(* IEC 61131-3 sources: Mizera_Tube/Plc (part 2) *)

(* ---- GasProp.plc ---- *)
*******************************************************************************
*   GASPROP.PLC
*   ESAutomotion
*   LASER machine - Proportional valve for cutting gas managment
*******************************************************************************
#funcdec "DynMng.plc"

VAR
#include "cnc.inc"

Appoggio:           BOOL;
KeepPropTest:       BOOL; * Prop. valve test keep
PropOutRange:       BOOL; * Gas pressure out of range
HbOutPress:         BOOL; * Hoerbiger feedback pressure out of range

PressCalcLinear:    DWORD; * Pressure calculated from linearization

AppPressCorrente:   DWORD; * Appoggio Pressione Corrente
MaxCurrPress:       DWORD; * Maximum pressure for current selected gas (mbar)
OutValvProp:        DWORD; * Prop valve setpoint pressure (mbar)
PressTol:           DWORD; * Pressure tolerance (mbar)
MinAllPressMbar:    DWORD; * Pressure min limit for alarm (mbar)
MaxAllPressMbar:    DWORD; * Pressure max limit for alarm (mbar)
TimeAlPress:        DWORD; * Delay for pressure alarm enable (ms)
ScaleBitIN:         DWORD; * Pressure input full scale in count
ScaleBitOUT:        DWORD; * Pressure output full scale in count
IA_Feedback_GAS_IN_BAR: DWORD; * Hoerbiger feedback pressure (bar)
PressMaxEvProp_APP: DWORD;

RTRIG_EnVal1:       TRIG;
RTRIG_EnVal1_G834:  TRIG;

HOERRB_CAL_REQ1     AT %SoftBtn2.10; * ANALOG HOERB CALIBRATION REQUEST BUTTON
HOERB_RESET_REQ   	AT %SoftBtn2.20; *(SoftBtn2.20) Hoerbiger reset button
TOF_RESET_HOERB:			TOF;			 * ANALOG HOERB RESET
RTRIG_RESET_HOERB:			R_TRIG;			 * ANALOG HOERB RESET REQUEST

RT_PVTST:           R_TRIG;
#defcom RT_PVTST.Q Imp. prop. valve test button
TRIG_CAL_HOERB:     TRIG; * Hoerbiger calibration request
#defcom TRIG_CAL_HOERB.Q Imp. Hoerbiger calibration request

TON_All_prop:       TON;
#defcom TON_All_prop.Q End of pressure alarm delay
TP_HOERB_CALIB:     TP;
#defcom TP_HOERB_CALIB.Q Time for Hoerbiger calibration request
TON_HOERB_CALIB2:   TON;
#defcom TON_HOERB_CALIB2.Q End delay for Hoerbiger calibration alarm
TON_FEEDBACK_GAS_IN: TON;
#defcom TON_FEEDBACK_GAS_IN.Q End of delay pressure check for Hoerbiger valve

GasCalc:           POINTS_INT_CALC;
GasCalc2:          POINTS_INT_CALC;

END_VAR

VAR_IN_OUT
#include "mem.inc"
END_VAR

#include "iol.inc"

*******************************************************************************
FUNCTION GasProp
*******************************************************************************

*******************************************************************************
*   Enable data writing
*   M300 or TstP14.14 (from TabLaser)
*******************************************************************************
CAL  RTRIG_EnVal1(CLK=EnValOut1)   ** (TstP14.14) Abilita Attuazione Valori Uscite
CAL  RTRIG_EnVal1_G834(CLK=EnValOut1_G834)   ** (TstP11.14) Abilita Attuazione Valori Uscite

LD   RTRIG_EnVal1.Q
OR   RTRIG_EnVal1_G834.Q
AND  PRGRUN_CN0                    ** M0.0 cn0.rc8.0  Programma in corso
ST   Appoggio

LD   %cn0.rc9                * Registro funzioni M canale 0
EQ   300
AND  %cn0.rc8.4              * Strobe funzioni M canale 0
OR   Appoggio
JMPCN COPYVAL

LD   %TabLsr0.L_CutPressure
ST   GasPressPgmSet                ** (LsPlc31) Gas pressure setpoint by program (mbar)

COPYVAL:

* Proportional valve type selection

LD   %config_machine4              ** LASER - Tipo gestione valv. prop. sul bus ECAT (0=DIWAL,1=HOERBIGER...)
EQ   0
AND  %config_machine2.0            ** LASER - Gestione valvola proporzionale sul bus ECAT
ST   GasPVDiwal                    ** M107.21 Cutting gas prop. valve type lanny diwal

LD   %config_machine4              ** LASER - Tipo gestione valv. prop. sul bus ECAT (0=DIWAL,1=HOERBIGER...)
EQ   1
AND  %config_machine2.0            ** LASER - Gestione valvola proporzionale sul bus ECAT
ST   GasPVHoerbiger                ** M107.22 Cutting gas prop. valve type hoerbiger

* Proportional valve test command

CAL  RT_PVTST(CLK=P_ValTestProp)   ** (LsGui18.9) Proportional valve test from setting page

LD   RT_PVTST.Q                    ** Imp. prop. valve test button
ANDN KeepPropTest                  ** Prop. valve test keep
S    KeepPropTest                  ** Prop. valve test keep
ST   Appoggio

LD   RT_PVTST.Q                    ** Imp. prop. valve test button
ANDN Appoggio
OR   PropTestRes                   ** M107.13 Proportional valve test reset from gas commands
OR   ProgRunForGas                 ** M107.10 Program running for gas managment
ORN  MACCHINA_OK                   ** M100.1  Macchina OK
OR   RESET_MACCHINA                ** M100.2  Reset macchina
R    KeepPropTest                  ** Prop. valve test keep

* Proportional valve enable conditions

LD   %config_machine29             ** Proportional valve manage only with OXYGEN
EQ   0
AND  O_O_EV_OR_ALLGAS              ** M90.15 Elettrovalvola apertura di almeno un gas
OR   O_O_EV_OPEN_O2                ** Elettrovalvola apertura Ossigeno
* La proporzionale viene disabilitata senza il ritardo alla disattivazione del program run
AND  (
LD   PRGRUN_CN0                    ** M0.0 cn0.rc8.0  Programma in corso
*ORN  ProgRunForGas                 ** M107.10 Program running for gas managment
)
OR   KeepPropTest                  ** Prop. valve test keep
OR   (
 LD   GAS_test                      ** M107.0 Test gas in progress for prop. valve
 AND  (
  LD   %config_machine29             ** Proportional valve manage only with OXYGEN
  EQ   0
      )
    )
OR  (
LD   GAS_test                      ** M107.0 Test gas in progress for prop. valve
 AND  (
   LD   %config_machine29             ** Proportional valve manage only with OXYGEN
   EQ   1
   AND  O_O_EV_OPEN_O2                ** Elettrovalvola apertura Ossigeno
   )
  )
OR   (
 LD   GAS_test
 OR   (
  LD   O_O_EV_OPEN_O2
  OR   O_O_EV_OPEN_N2
  OR   O_O_EV_OPEN_ARIA
  )
  AND  (
  LD   %config_machine29             ** Proportional valve manage only with OXYGEN
  EQ   2
 )
)
ANDN GAS_prun_close_propv
ST   GasPropEnabFromV              ** M107.23 Gas prop. valve enable from valve configuration

*******************************************************************************
* Pressure limit for selected gas
*******************************************************************************

* Pressure limit for oxygen

LD   0
ST   MaxCurrPress                  ** Maximum pressure for current selected gas (mbar)

LD   O_O_EV_OPEN_O2                ** Elettrovalvola apertura Ossigeno
JMPCN MP_OXIGEN

LD   PressMaxOssigeno              ** (rLsGui12)Pressione massima Ossigeno
ST   PressMaxEvProp_APP
ST   MaxCurrPress                  ** Maximum pressure for current selected gas (mbar)

MP_OXIGEN:

* Pressure limit for nitrogen

LD   O_O_EV_OPEN_N2                ** Elettrovalvola apertura Azoto
JMPCN MP_NITROGEN

LD   PressMaxAzoto                 ** (rLsGui13)Pressione massima Azoto
ST   MaxCurrPress                  ** Maximum pressure for current selected gas (mbar)

LD   PressMaxEvProp                ** (rLsGui11)Pressione massima valvola proporzionale
ST   PressMaxEvProp_APP

MP_NITROGEN:

* Pressure limit for cutting air

LD   O_O_EV_OPEN_ARIA              ** Elettrovalvola apertura Aria taglio
JMPCN MP_AIR

LD   PressMaxAria                  ** (rLsGui14)Pressione massima Aria
ST   MaxCurrPress                  ** Maximum pressure for current selected gas (mbar)

LD   PressMaxEvProp                ** (rLsGui11)Pressione massima valvola proporzionale
ST   PressMaxEvProp_APP

MP_AIR:

*******************************************************************************
* SETPOINT GAS PRESSURE SELECTION
*******************************************************************************
LD   0
ST   OutValvProp                   ** Prop valve setpoint pressure (mbar)

LD   GasPropEnabFromV              ** M107.23 Gas prop. valve enable from valve configuration
ANDN RETRACERUN                    ** M0.11 Ciclo di retrace in Run
JMPCN END_PRESS_UPD

* Gas pressure for Z up simulation

LD   GasEnabOnZUp                  ** M107.11 Gas enable conditions on Z up simulation
JMPCN Z_up_test

LD   %TabLsr0.L_CutPressure
ST   OutValvProp                   ** Prop valve setpoint pressure (mbar)

JMP  END_PRESS_UPD

Z_up_test:
LD   %LaserShootOn
JMPCN Z_up_test2

LD   %LsrGest0.ShootGasPress
ST   OutValvProp                   ** Prop valve setpoint pressure (mbar)

JMP  CHK_PROP_LIM

Z_up_test2:
* Gas pressure for PURGE or GAS test

LD   SPURGOrun                     ** M107.2 Gas purge in progress
JMPCN END_PURGE

LD   PressSpurgoGas                ** (rLsGui16)Pressione spurgo Gas
ST   OutValvProp                   ** Prop valve setpoint pressure (mbar)

JMP  CHK_PROP_LIM

END_PURGE:

LD   GAS_test                      ** M107.0 Test gas in progress for prop. valve
OR   KeepPropTest                  ** Prop. valve test keep
JMPCN END_PRGTST

LD   PressTestGas                  ** (rLsGui15)Pressione test Gas
ST   OutValvProp                   ** Prop valve setpoint pressure (mbar)

* Pressure limits for test/purge

CHK_PROP_LIM:

LD   OutValvProp                   ** Prop valve setpoint pressure (mbar)
GT   30000
JMPCN LIM_SUP

LD   30000
ST   OutValvProp                   ** Prop valve setpoint pressure (mbar)

JMP  LIM_INF

LIM_SUP:

LD   OutValvProp                   ** Prop valve setpoint pressure (mbar)
LT   50
JMPCN LIM_INF

LD   50
ST   OutValvProp                   ** Prop valve setpoint pressure (mbar)

LIM_INF:

* With gas valve ON, check the pressure limits for selected gas
LD   O_O_EV_OR_ALLGAS              ** M90.15 Elettrovalvola apertura di almeno un gas
JMPC CHK_PRESS_LIM

JMP  END_PRESS_UPD

END_PRGTST:

* Air pressure for APA

LD   AirEnabForAPA                 ** M107.12 Cutting air enable for APA cycle
JMPCN NoApaRun

LD   %config_machine23             ** Pressione ARIA per gestione APA
ST   OutValvProp                   ** Prop valve setpoint pressure (mbar)
JMP  END_PRESS_UPD

NoApaRun:

* Gas pressure for program execution

LD   GasPressPgmSet                ** (LsPlc31) Gas pressure setpoint by program (mbar)
ST   OutValvProp                   ** Prop valve setpoint pressure (mbar)

* Pressure limit for selected gas

CHK_PRESS_LIM:

LD   OutValvProp                   ** Prop valve setpoint pressure (mbar)
GT   MaxCurrPress                  ** Maximum pressure for current selected gas (mbar)
JMPCN END_PRESS_UPD

LD   MaxCurrPress                  ** Maximum pressure for current selected gas (mbar)
ST   OutValvProp                   ** Prop valve setpoint pressure (mbar)

END_PRESS_UPD:

LD   OutValvProp                   ** Prop valve setpoint pressure (mbar)
ST   SetOutPress                   ** (LsPlc38) Setpoint output pressure (mbar)

LD   SetOutPress                   ** (LsPlc38) Setpoint output pressure (mbar)
MUL  145                           * 14.5 PSI = 1 bar
DIV  1000
ST   SetPressPSI                   ** (LsPlc39) Setpoint output pressure (PSI*10)

********************************************************************************
* OUTPUT GAS PRESSURE COMMAND                                                  *
********************************************************************************
LD   GasPVDiwal                    ** M107.21 Cutting gas prop. valve type lanny diwal
JMPCN no_diwal_valve

LD   GAS_test                      ** M107.0 Test gas in progress for prop. valve
OR (
LD   GAS_prun                      ** M107.1 Cutting gas active from part program
ANDN GAS_prun_close_propv
)
OR   KeepPropTest                  ** Prop. valve test keep
ST   O_O_GAS_ECAT_TYPE0_ENAB       ** Enable proportional valve on bus ecat

no_diwal_valve:
LD   GasPVHoerbiger                ** M107.22 Cutting gas prop. valve type hoerbiger
OR   GasPVDiwal                    ** M107.21 Cutting gas prop. valve type lanny diwal
JMPC NoAnalogV

***************************************
*   ANALOG valve
***************************************
* Selection 12 or 16 bits output resolution

LD   BitOutValvProp                ** (rLsPlc42) Numero bit x uscita valvola prop.
EQ   0
JMPCN l11bitOut

LD   4095
ST   ScaleBitOUT                   ** Pressure output full scale in count

JMP  ComBitOut

l11bitOut:
LD   BitOutValvProp                ** (rLsPlc42) Numero bit x uscita valvola prop.
EQ   2
JMPCN l16bitOut

LD   2047
ST   ScaleBitOUT                   ** Pressure output full scale in count

JMP  ComBitOut

l16bitOut:
LD   32767
ST   ScaleBitOUT                   ** Pressure output full scale in count

ComBitOut:

NoAnalogV:
***********************************************************
* Gases Linearization
***********************************************************
LD   EnabGasOutByGraph	     			     **(rLsGui25.0) PLC option for enabling the graph (Pressure-voltage)
JMPCN NO_LINEAR

        LD   O_O_EV_OPEN_ARIA
        OR   O_O_EV_OPEN_N2
        JMPCN NO_HP_VALVE
             LD   SetOutPress                   ** (LsPlc38) Setpoint output pressure (mbar)
             ST   GasCalc2.xPercSpeed            * Speed percentual value

             LD   1
             ST   GasCalc2.xCutLineInd           * cut line index (initial value 1 to 10)

             LD   45
             ST   GasCalc2.xCodTec               * Tecnology 0=duty 1=power 2=frequency

             CAL  GasCalc2

             LD   GasCalc2.yResult               * Result
             ST   PressCalcLinear
        NO_HP_VALVE:

        LD   O_O_EV_OPEN_O2
        JMPCN ONLY_O2_VALVE
             LD   SetOutPress                   ** (LsPlc38) Setpoint output pressure (mbar)
             ST   GasCalc.xPercSpeed            * Speed percentual value

             LD   1
             ST   GasCalc.xCutLineInd           * cut line index (initial value 1 to 10)

             LD   40
             ST   GasCalc.xCodTec               * Tecnology 0=duty 1=power 2=frequency

             CAL  GasCalc

             LD   GasCalc.yResult               * Result
             ST   PressCalcLinear
        ONLY_O2_VALVE:

		 ***************************************
         *   Gas=funz(angle)
         *   #CDL
         ***************************************
         LD   PRGRUN_CN0
         ANDN PRGSTOP_CN0
         AND (
         LD   %uvHeads0.uvhCommand1
         EQ   4                              * Cutting phase
         )
         AND  %LSRPlcOp0.3
         JMPCN no_corr_gas_linear
               LD   PressCalcLinear
               ADD (
               LD   PressCalcLinear
               MULDIV(M=%TsCutDataLinear.CDL_Pressure,D=100000) * 100 %
               )
               ST   PressCalcLinear
         no_corr_gas_linear:

        *---------------------
        *   DIWAL
        *---------------------
        LD   GasPVDiwal                         ** M107.21 Cutting gas prop. valve type lanny diwal
        JMPCN NoLin1
             LD   PressCalcLinear               ** (LsPlc38) Setpoint output pressure (mbar)
             ***DIV  10000
             ST   OA_GAS_ECAT_TYPE0             ** Gas valve on bus ecat
        NoLin1:

        *---------------------
        *   HOERBIGER
        *---------------------
        LD   GasPVHoerbiger                     ** M107.22 Cutting gas prop. valve type hoerbiger
        JMPCN NoLin2
             LD   PressCalcLinear               ** (LsPlc38) Setpoint output pressure (mbar)
             ***DIV  10000
             ST   O_OA_GAS_HOERB
        NoLin2:

        *---------------------
        *   ANALOG
        *---------------------
        LD   PressCalcLinear                   ** (LsPlc38) Setpoint output pressure (mbar)
        MUL  ScaleBitOUT                   ** Pressure output full scale in count
        DIV  PressMaxEvProp_APP
        ST   OA_GAS                        ** Gas analog valve

JMP ComValv_

NO_LINEAR:

         ***************************************
         *   Gas=funz(angle)
         *   #CDL
         ***************************************
         LD   PRGRUN_CN0
         ANDN PRGSTOP_CN0
         AND (
         LD   %uvHeads0.uvhCommand1
         EQ   4                              * Cutting phase
         )
         AND  %LSRPlcOp0.3
         JMPCN no_corr_gas
              LD   PressCalcLinear
              ADD (
              LD   PressCalcLinear
              MULDIV(M=%TsCutDataLinear.CDL_Pressure,D=100000) * 100 %
              )
              ST   PressCalcLinear
         no_corr_gas:

         *---------------------
         *   DIWAL
         *---------------------
         LD   GasPVDiwal                    ** M107.21 Cutting gas prop. valve type lanny diwal
         JMPCN NoLin10
              LD   SetOutPress              ** (LsPlc38) Setpoint output pressure (mbar)
              ST   OA_GAS_ECAT_TYPE0        ** Gas valve on bus ecat
         NoLin10:
         *---------------------
         *   HOERBIGER
         *---------------------
         LD   GasPVHoerbiger                ** M107.22 Cutting gas prop. valve type hoerbiger
         JMPCN NoLin20
              LD   SetOutPress              ** (LsPlc38) Setpoint output pressure (mbar)
              ST   O_OA_GAS_HOERB
         NoLin20:

         *---------------------
         *   ANALOG
         *---------------------
         LD   SetOutPress                   ** (LsPlc38) Setpoint output pressure (mbar)
         MUL  ScaleBitOUT                   ** Pressure output full scale in count
         DIV  PressMaxEvProp_APP
         ST   OA_GAS                        ** Gas analog valve

ComValv_:

**********************************************************************
* HOERBIGER valve calibration
**********************************************************************
LD   GasPVHoerbiger                ** M107.22 Cutting gas prop. valve type hoerbiger
JMPCN NoHber

CAL  TRIG_CAL_HOERB(CLK=HOERRB_CAL_REQ) ** Hoerbiger calibration request

CAL  TP_HOERB_CALIB(IN:=TRIG_CAL_HOERB.Q, PT=7000) ** Imp. Hoerbiger calibration request

LD   TP_HOERB_CALIB.Q              ** Time for Hoerbiger calibration request
ST   O_O_CALIB_REQ_HOERB           ** Hoerbiger: calibration request

LDN  I_I_HOERBIGER_READY           ** Hoerbiger ready on bus ecat
ST   Appoggio

CAL  TON_HOERB_CALIB2(IN:=Appoggio,PT:=15000)

LD   TON_HOERB_CALIB2.Q            ** End delay for Hoerbiger calibration alarm
ST   %PLCerr7.8                   * hoerbiger calibration error

NoHber:

*------------------------------------------------------------------------------*
* CURRENT GAS PRESSURE READING
*------------------------------------------------------------------------------*

LD   GasPVDiwal                    ** M107.21 Cutting gas prop. valve type lanny diwal
JMPCN no_lanny_diwal

* Diwal valve pressure reading

LD   IA_FBACK_ECAT_TYPE0           ** Gas proportional valve feedback on bus ecat
ST   AppPressCorrente              ** Appoggio Pressione Corrente

JMP  ComValv

no_lanny_diwal:

LD   GasPVHoerbiger                ** M107.22 Cutting gas prop. valve type hoerbiger
JMPCN no_hoerbiger

* Hoerbiger valve pressure reading

LD   IA_Feedb_HOERB_GAS_OUT        ** Hoerbiger gas proportional valve feedback (OUTPUT)
ST   AppPressCorrente              ** Appoggio Pressione Corrente
JMP  ComValv

no_hoerbiger:

* Selection 12 or 16 bits input resolution

LD   BitInValvProp                 ** (rLsPlc39) Numero bit x feedback valvola prop.
EQ   0
JMPCN l16bitIn

LD   4095
ST   ScaleBitIN                    ** Pressure input full scale in count
JMP  ComBitIn

l16bitIn:

LD   BitInValvProp                 ** (rLsPlc39) Numero bit x feedback valvola prop.
EQ   1
JMPCN l16bitInFull

LD   32767
ST   ScaleBitIN                    ** Pressure input full scale in count
JMP  ComBitIn

l16bitInFull:

LD   65535
ST   ScaleBitIN                    ** Pressure input full scale in count

ComBitIn:

* Analog valve pressure reading

LD   IA_Feedback_GAS_OUT           ** Gas proportional valve feedback (OUTPUT)
MUL  PressMaxEvProp_APP
DIV  ScaleBitIN                    ** Pressure input full scale in count
ST   AppPressCorrente              ** Appoggio Pressione Corrente

LD   %config_machine29             ** Proportional valve manage only with OXYGEN
EQ   2
JMPCN AIRO2_O2_SMCS
     LD   IA_Feedback_GAS_OUT      ** (IW20)Feedback valvola proporzionale gas di taglio Output
     SUB  819
	 MUL  PressMaxEvProp_APP
     DIV  (
     LD   ScaleBitIN
     SUB  819
     )
     ST   AppPressCorrente         ** Appoggio Pressione Corrente

     * Avoid negative value visualizzation
     LD   AppPressCorrente
     LT   0
     JMPCN no_force_zero
     LD   0
     ST   AppPressCorrente
     no_force_zero:
AIRO2_O2_SMCS:

ComValv:

LD   AppPressCorrente              ** Appoggio Pressione Corrente
ST   PressCorrente                 ** (LsPlc35) Pressione Corrente (mbar)

LD   PressCorrente                 ** (LsPlc35) Pressione Corrente (mbar)
MUL  145                           * 14.5 PSI = 1 bar
DIV  1000
ST   CurPressPSI                   ** (LsPlc34) Current gas pressure (PSI*10)

****************************************************************************************************
* GAS PRESSURE OUT OF RANGE ALARM
****************************************************************************************************
LD   SetOutPress                   ** (LsPlc38) Setpoint output pressure (mbar)
MUL  FinestraAllPress              ** (rLsGui18)Finestra allarme pressione da pagina "Gas" in %
DIV  100
ST   PressTol                      ** Pressure tolerance (mbar)

LD   SetOutPress                   ** (LsPlc38) Setpoint output pressure (mbar)
ADD  PressTol                      ** Pressure tolerance (mbar)
ST   MaxAllPressMbar               ** Pressure max limit for alarm (mbar)

LD   SetOutPress                   ** (LsPlc38) Setpoint output pressure (mbar)
SUB  PressTol                      ** Pressure tolerance (mbar)
ST   MinAllPressMbar               ** Pressure min limit for alarm (mbar)

LD   MinAllPressMbar               ** Pressure min limit for alarm (mbar)
LT   0
JMPCN NoZeroMin

LD   0
ST   MinAllPressMbar               ** Pressure min limit for alarm (mbar)

NoZeroMin:

LD   PressCorrente                 ** (LsPlc35) Pressione Corrente (mbar)
GE   MinAllPressMbar               ** Pressure min limit for alarm (mbar)
AND (
LD   PressCorrente                 ** (LsPlc35) Pressione Corrente (mbar)
LE   MaxAllPressMbar               ** Pressure max limit for alarm (mbar)
)
OR   (
LD   FinestraAllPress              ** (rLsGui18)Finestra allarme pressione da pagina "Gas" in %
EQ   0
)
AND  GasPropEnabFromV              ** M107.23 Gas prop. valve enable from valve configuration
ST   PressGasOk                    ** M107.20 Gas pressure in range

LD   GasPropEnabFromV              ** M107.23 Gas prop. valve enable from valve configuration
ANDN PressGasOk                    ** M107.20 Gas pressure in range
ANDN SPURGOrun                     ** M107.2 Gas purge in progress
ST   PropOutRange                  ** Gas pressure out of range

LD   TimeMaxAllPress               ** (rLsGui19)Tempo Ritardo allarme pressione da pagina "Gas"
MUL  1000
ST   TimeAlPress                   ** Delay for pressure alarm enable (ms)

CAL  TON_All_prop(IN=PropOutRange,PT=TimeAlPress) ** Gas pressure out of range

LD   TON_All_prop.Q                ** End of pressure alarm delay
S    %PLCerr5.14                  ** PLC Err 174 Pressione valvola proporzionale fuori range

LD   RESET_ALLARMI                 ** M100.4  Cancellazione allarmi attiva
OR   Pul_Start                     ** (gPlc0.1)Start pushbutton
R    %PLCerr5.14                  ** PLC Err 174 Pressione valvola proporzionale fuori range

**********************************************************************
* Control of input gasses (AIR / O2 / N2) with Hoerbiger input valve
**********************************************************************

LD   IA_Feedback_GAS_IN_DIG        ** Hoerbiger gas proportional valve feedback (INPUT)
ST   IA_Feedback_GAS_IN_BAR        ** Hoerbiger feedback pressure (bar)

LD   O_O_EV_OR_ALLGAS              ** M90.15 Elettrovalvola apertura di almeno un gas
AND  PRGRUN_CN0                    ** M0.0 cn0.rc8.0  Programma in corso
AND  GasPVHoerbiger                ** M107.22 Cutting gas prop. valve type hoerbiger
ST   Appoggio

CAL  TON_FEEDBACK_GAS_IN(IN:=Appoggio,PT:=Delay_Press_Check) ** (rLsGui21) Delay_Press_Check

LD   MaxCurrPress                  ** Maximum pressure for current selected gas (mbar)
SUB  IA_Feedback_GAS_IN_BAR        ** Hoerbiger feedback pressure (bar)
GT   Diff_Limit_Pres               ** (rLsGui22) Input limit difference pressure
AND  TON_FEEDBACK_GAS_IN.Q         ** End of delay pressure check for Hoerbiger valve
ANDN SPURGOrun                     ** M107.2 Gas purge in progress
ST   HbOutPress                    ** Hoerbiger feedback pressure out of range

LD   HbOutPress                    ** Hoerbiger feedback pressure out of range
AND  O_O_EV_OPEN_ARIA              ** Elettrovalvola apertura Aria taglio
S    %PLCerr7.12                    ** Hoerbiger low air pressure

LD   HbOutPress                    ** Hoerbiger feedback pressure out of range
AND  O_O_EV_OPEN_N2                ** Elettrovalvola apertura Azoto
S    %PLCerr7.13                    ** Hoerbiger low nitrogen pressure

LD   HbOutPress                    ** Hoerbiger feedback pressure out of range
AND  O_O_EV_OPEN_O2                ** Elettrovalvola apertura Ossigeno
S    %PLCerr7.14                    ** Hoerbiger low oxigen pressure

LD   Pul_Reset                     ** (gPlc0.3)Reset pushbutton
OR   EMERGENZA_PLC_CN              ** M100.0  Emergenza da PLC o da CN
OR   Pul_Start                     ** (gPlc0.1)Start pushbutton
R    %PLCerr7.12                    ** Hoerbiger low air pressure
R    %PLCerr7.13                    ** Hoerbiger low nitrogen pressure
R    %PLCerr7.14                    ** Hoerbiger low oxigen pressure

LD   %PLCerr7.12                   ** Hoerbiger low air pressure
OR   %PLCerr7.13                   ** Hoerbiger low nitrogen pressure
OR   %PLCerr7.14                   ** Hoerbiger low oxigen pressure
ST   Hold_gas_refill               ** M107.24 Hoerbiger insufficient gas pressure

****************************************************************************************************
* Segnalazioni su pagina video
****************************************************************************************************

LD   GAS_test                      ** M107.0 Test gas in progress for prop. valve
OR   KeepPropTest                  ** Prop. valve test keep
AND  GasPropEnabFromV              ** M107.23 Gas prop. valve enable from valve configuration
ST   GasTestLED                    ** (LsPlc11.10) LED Comando TEST Valvola prop.

**********************************************************************
* HOERBIGER RESET
**********************************************************************

LD   HOERB_RESET_REQ			*(SoftBtn2.20) Hoerbiger reset button
ANDN %PLCmsg7.1					*Hoerbiger calibration not running
ST   Appoggio

CAL  RTRIG_RESET_HOERB(CLK=Appoggio)
CAL  TOF_RESET_HOERB(IN:=RTRIG_RESET_HOERB.Q, PT=3000)

LD   TOF_RESET_HOERB.Q
ST   O_O_HOER_RESET

END_FUNCTION

(* ---- GestAssi.plc ---- *)
*******************************************************************************
*   GESTASSI.PLC
*   ESAutomotion
*   LASER machine
*******************************************************************************
VAR
#include "Cnc.inc"

TOF_AxStop: TOF;    *Ritardo diseccitazione Assi Fermi

END_VAR

VAR_IN_OUT
#include "mem.inc"
END_VAR

#include "Iol.inc"

*******************************************************************************
*   * Gestione Segnali assi
*******************************************************************************
FUNCTION Gest_Assi

*******************************************************************************
*   Gestione segnali asse X1
*******************************************************************************
* Richiesta ordine di moto asse X1
LD   %ax27.ra3.10           * Anello di regolazione attivo
AND  %ax27.ra3.13           * Ordine di moto
ST   Ordine_Moto_X1                ** M71.0 Ordine di moto asse X1

* Moto asse X+
LD   Ordine_Moto_X1                ** M71.0 Ordine di moto asse X1
ANDN %ax27.ra3.0            * Asse fermo teorico
AND  %ax27.ra3.2            * Direzione moto asse+
ANDN AsseX1_Moto_neg               ** M71.2 Asse X1 in moto -
ST   AsseX1_Moto_pos               ** M71.1 Asse X1 in moto +

* Moto asse X-
LD   Ordine_Moto_X1                ** M71.0 Ordine di moto asse X1
ANDN %ax27.ra3.0            * Asse fermo teorico
ANDN %ax27.ra3.2            * Direzione moto asse+
ANDN AsseX1_Moto_pos               ** M71.1 Asse X1 in moto +
ST   AsseX1_Moto_neg               ** M71.2 Asse X1 in moto -

*******************************************************************************
*   Gestione segnali asse Y1
*******************************************************************************
* Richiesta ordine di moto asse Y1
LD   %ax28.ra3.10           * Anello di regolazione attivo
AND  %ax28.ra3.13           * Ordine di moto
ST   Ordine_Moto_Y1                ** M71.8 Ordine di moto asse Y1

* Moto asse Y+
LD   Ordine_Moto_Y1                ** M71.8 Ordine di moto asse Y1
ANDN %ax28.ra3.0            * Asse fermo teorico
AND  %ax28.ra3.2            * Direzione moto asse+
ANDN AsseY1_Moto_neg               ** M71.10 Asse Y1 in moto -
ST   AsseY1_Moto_pos               ** M71.9 Asse Y1 in moto +

* Moto asse Y-
LD   Ordine_Moto_Y1                ** M71.8 Ordine di moto asse Y1
ANDN %ax28.ra3.0            * Asse fermo teorico
ANDN %ax28.ra3.2            * Direzione moto asse+
ANDN AsseY1_Moto_pos               ** M71.9 Asse Y1 in moto +
ST   AsseY1_Moto_neg               ** M71.10 Asse Y1 in moto -

*******************************************************************************
*   Gestione segnali asse Z1
*******************************************************************************
* Richiesta ordine di moto asse Z1
LD   %ax29.ra3.10           * Anello di regolazione attivo
AND  %ax29.ra3.13           * Ordine di moto
ST   Ordine_Moto_Z1                ** M71.16 Ordine di moto asse Z1

* Moto asse Z+
LD   Ordine_Moto_Z1                ** M71.16 Ordine di moto asse Z1
ANDN %ax29.ra3.0            * Asse fermo teorico
AND  %ax29.ra3.2            * Direzione moto asse+
ANDN AsseZ1_Moto_neg               ** M71.18 Asse Z1 in moto -
ST   AsseZ1_Moto_pos               ** M71.17 Asse Z1 in moto +

* Moto asse Z-
LD   Ordine_Moto_Z1                ** M71.16 Ordine di moto asse Z1
ANDN %ax29.ra3.0            * Asse fermo teorico
ANDN %ax29.ra3.2            * Direzione moto asse+
ANDN AsseZ1_Moto_pos               ** M71.17 Asse Z1 in moto +
ST   AsseZ1_Moto_neg               ** M71.18 Asse Z1 in moto -

*******************************************************************************
*   Posizione sicura Asse Z per moto assi
*******************************************************************************
LD   %ax29.ra4              ** Quota asse Z
GT   %LSRCostK48            ** Valore quota sicurezza asse Z in pagina video
AND  %ax29.ra3.14           * ra3.14  Asse Z tarato
ST   Ax_Z1_posiz_OK                ** M74.7 Asse Z1 in posizione di sicurezza

LD   MACCH_IN_AUTO                 ** M100.25 SELEZIONE MACCHINA IN AUTOMATICO
ANDN PRGRUN_CN0                    ** M0.0 cn0.rc8.0  Programma in corso
OR   MACCH_IN_MANUALE              ** M100.24 SELEZIONE MACCHINA IN MANUALE
ANDN PLC_SEL_REF                   ** ui16.1 Selezione Modo REF da Plc
ANDN Ax_Z1_posiz_OK                ** M74.7 Asse Z1 in posizione di sicurezza
ST   BlcAvX1_Z1_no_OK              ** M74.2 Blocco avanz. asse X1 per Asse Z1 non posiz. OK
ST   BlcAvY1_Z1_no_OK              ** M74.5 Blocco avanz. asse Y per Asse Z non posiz. OK

LD   BlcAvX1_Z1_no_OK              ** M74.2 Blocco avanz. asse X1 per Asse Z1 non posiz. OK
AND  %ax27.ra3.13           ** X1 Ordine di moto +\-
ST   %PLCmsg4.12            ** Plc Msg 140 Blocco Asse X1:Asse Z1 non in posizione di sicurezza

LD   BlcAvY1_Z1_no_OK              ** M74.5 Blocco avanz. asse Y per Asse Z non posiz. OK
AND  %ax28.ra3.13           * Y1 Ordine di moto +\-
ST   %PLCmsg4.16            ** Plc Msg 144 Blocco Asse Y1:Asse Z1 non in posizione di sicurezza

*******************************************************************************
*   Blocco Avanzamento X1/Y1: Sensore capacitivo in contatto con la lamiera
*******************************************************************************
LD   %PLCerr5.4             **PLC Err 164 Tip touch (A11=1, A14=0, A15=0 in normal operation)
OR   %PLCerr5.5             **PLC Err 165 Body touch (A11=1, A14=1, A15=0 in normal operation)
ANDN GEN_REF_RUN                   ** M100.16 Ciclo di Reference GENERALE in corso
ST   BlcAvX1_Sens_Capac            ** M74.3 Blocco avanz. asse X1 Sens. Capacitivo in contatto con la lamiera
ST   BlcAvY1_Sens_Capac            ** M74.6 Blocco avanz. asse Y Sens. Capacitivo in contatto con la lamiera

*******************************************************************************
*   Blocco avanzamento X1/Y1
*******************************************************************************
LD   BL_AV_ASSI_X_OVR              ** M74.8 Blocco avanzamento assi dopo Override=0 o NC_STOP
ANDN PRGSTOP_CN0                   ** (cn0.rc8.1)  Programma interrotto CN0
OR   BlcAvX1_Z1_no_OK              ** M74.2 Blocco avanz. asse X1 per Asse Z1 non posiz. OK
OR   BlcAvX1_Sens_Capac            ** M74.3 Blocco avanz. asse X1 Sens. Capacitivo in contatto con la lamiera
OR   BlcAvY1_Sens_Capac            ** M74.6 Blocco avanz. asse Y Sens. Capacitivo in contatto con la lamiera
ST   BlcAvX1_user                  ** M74.0 Blocco avanzamento asse X1 da user.plc
ST   BlcAvY1_user                  ** M74.4 Blocco avanzamento asse Y da user.plc

****************************************************************************************************
*   Segnale Assi Fermi
****************************************************************************************************
CAL  TOF_AxStop(IN=AxStopSincGRP,PT=50) ** Ritardo diseccitazione Assi Fermi

LD   TOF_AxStop.Q
ST   AxStop_ForUser                ** (gPlc13.14) Info Assi fermi a User

END_FUNCTION

(* ---- IOConfig.plc ---- *)
*******************************************************************************
*   IOCONFIG.PLC
*   ESAutomotion
*   LASER machine
*******************************************************************************
#funcdec "res_ipg.plc"
#funcdec "LsrGest.plc"
#funcdec "CAP_Prec.plc"
#funcdec "FocProco.plc"

VAR
#include "Cnc.inc"
#include "Iof.inc"       * I/O Applicativo
END_VAR

VAR_IN_OUT
#include "mem.inc"
END_VAR

#include "Iol.inc"
#include "res_ipg.inc"
#include "LsrGest.inc"
#include "Cap_Prec.inc"
#include "foc_prec.inc"
#include "Aspiraz.inc"
#include "nLight.inc"

*#include "zVar.inc"

VAR
TM_offLSR:                       TOF;
TM_OnLSR:                        TON;
TM_StartButton:                   TP;
AppStartLSR:                    BOOL;
GuardDoorAutoUp:                BOOL;
GuardDoorAutoDwn:               BOOL;
RTRIG_A1_LASER_REQ:           R_TRIG;
TOF_A1_LASER_REQ:                TOF;

TP_Fence:                         TP;
FTRIG_Fence:                  F_TRIG;
R_TRIG_Door_Up_Gui_1:         R_TRIG;
R_TRIG_Door_Down_Gui_1:       R_TRIG;
R_TRIG_Door_Up_Gui_2:         R_TRIG;
R_TRIG_Door_Down_Gui_2:       R_TRIG;
END_VAR

*******************************************************************************
*   I/O CONFIGURATION (INPUT)
*******************************************************************************
FUNCTION INP_CONFIG

***************************************
*   GENERIC
***************************************
LDN  I_EMERGENZA
S    I_I_EMERGENZA               * Machine OK (no EMERG.)

LD   Pul_Reset
R    I_I_EMERGENZA

LD   I_CHILLER_ERR				* Chiller error
ANDN %LSRPlcOp0.8
ST   I_I_CHILLER_ERR
ST   %PLCerr6.0

LD   I_ASPIRATORE_OK
ST   I_I_ASPIRATORE_OK

***
*** *Comandi operatore
*** *----------------------------
LD  I_PUL_START
ST  I_I_PUL_START               * Start
LD  I_PUL_STOP
ST  I_I_PUL_STOP                * Stop
LD  I_PUL_RESET
ST  I_I_PUL_RESET               * Reset
***
*** *Hold macchina
*** *----------------------------
***  LD  M_HoldAlarmMac              *Hold macchina per allarme
***  ST  CMD_HOLD_MAC                * M206.0 Hold (CH0, CH3)
***
*** *Hold assi
*** *----------------------------
***  LD  M_HoldAx_X
***  ST  CMD_HOLDMOVING_CH3.0
***  LD  M_HoldAx_Y
***  ST  CMD_HOLDMOVING_CH3.1
***  LD  M_HoldAx_Z
***  ST  CMD_HOLDMOVING_CH3.2
*** LD  M_HoldAx_U
*** ST  CMD_HOLDMOVING_CH3.3
***  LD  M_HoldAx_B
***  ST  CMD_HOLDMOVING_CH3.7
***  LD  M_HoldAx_Cm
***  ST  CMD_HOLDMOVING_CH3.8
***
***  LD  M_HoldAx_Cs
***  ST  CMD_HOLDMOVING_CH5.8

 *Drives ok
 *----------------------------

*************************************************
*   GAS
*************************************************
 *Ingresso analogica
 *----------------------------
  LD  %ecat_ring0.EcatNode20.EcMDPIn1
  ST  IA_FBACK_ECAT_TYPE0

 *Ingresso digitale
 *----------------------------
  LD  I_PRESSIONE_ARIA_IMPIANTO
  ST  I_I_PRESSIONE_ARIA_IMPIANTO * Pressione aria Impianto OK

  LD  I_PRESSIONE_N2
  ST  I_I_PRESSIONE_N2            * Pressione Azoto OK

  LD  I_PRESSIONE_O2
  ST  I_I_PRESSIONE_O2            * Pressione Ossigeno OK

  LD  I_PRESSIONE_ARIA
  OR(
   LD %rLsGui14
   LE 0
  )
  ST  I_I_PRESSIONE_ARIA          * Pressione Aria di taglio OK

  LD  I_PRESSIONE_ARIA_BANCO      * PLCFLAGS.1  Flag sempre stato on
  ST  I_I_PRESSIONE_ARIA_BANCO    * Pressione aria Banco OK

* HOERBIGER VALVE

LD   I_IA_Feedb_HOERB_GAS_OUT
ST   IA_Feedb_HOERB_GAS_OUT       * Hoerbiger gas proportional valve feedback (OUTPUT)

LD   I_HOERBIGER_READY          * Hoerbiger ready on bus ecat
ST   I_I_HOERBIGER_READY          * Hoerbiger ready on bus ecat

*************************************************
*   RESONATOR (IPG)
*************************************************
PATH %Resonator[0]
PATH %LsrGest[0]

* Gestione laser IPG YSL
***************************************
LD   %config_machine28
EQ   0
JMPCN NoLSR_IPG_YLS

 *Ingressi digitali
 *----------------------------
  LD   I_LSR_READY
  ST   I_B1_LASER_READY           ** IPG Laser internal main power supply ON (Aux Power ON)

  LD   I_LSR_WARNING
  ST   I_B13_AVVERTENZA           ** IPG WARNING OUT

  LD   I_LSR_ERROR
  ST   I_B4_LASER_ERROR           ** IPG YLS YLR Laser in Alarm status

  LD   I_LSR_GUIDE_ON
  ST   I_B5_LASER_GUIDE           ** IPG Laser guida ON

  LD   I_LSR_EMISSION_ON
  ST   I_B2_EMISSION_ON           ** IPG Emission ON

  LD   ALWAYS_ONE
  ST   I_B7_LASER_ASSIGNED        ** IPG Laser ASSIGNED

  LD   ALWAYS_ONE
  ST   I_B8_POWER_SUPPLY          ** IPG power supply status

  LD   ALWAYS_ONE
  ST   I_B6_ANALOG_CONTROL        ** IPG Controllo analogico ON

***************************************
NoLSR_IPG_YLS:

*Gestione laser IPG YSR - RACK
***************************************
LD   %config_machine28
EQ   1
JMPCN NoLSR_IPG_YLR

 *Ingressi digitali
 *----------------------------
  LD   %PLCFLAGS.1
  ST   I_B1_LASER_READY              ** IPG Laser internal main power supply ON (Aux Power ON)

  LDN  I_LSR_READY
  AND  I_LSR_LASER_ON
  ST   I_B4_LASER_ERROR              ** IPG YLS YLR Laser in Alarm status

  LD   I_LSR_EMISSION_ON
  ST   I_B2_EMISSION_ON              ** IPG Emission ON

  LD   %PLCFLAGS.1
  ST   I_B7_LASER_ASSIGNED           ** IPG Laser ASSIGNED

  LD   ALWAYS_ONE
  ST   I_B8_POWER_SUPPLY             ** IPG power supply status

 *Ingressi simulati
 *----------------------------
  LD   %PLCFLAGS.0
  ST   I_B13_AVVERTENZA              ** IPG WARNING OUT

  LD   O_A6_ANALOG_CONTROL
  AND  I_B8_POWER_SUPPLY             ** IPG power supply status
  ST   I_B6_ANALOG_CONTROL           ** IPG Controllo analogico ON

  LD   O_A5_GUIDE_LASER
  AND  I_B8_POWER_SUPPLY             ** IPG power supply status
  ST   I_B5_LASER_GUIDE              ** IPG Laser guida ON

 *SEGNALI NON GESTITI
 *----------------------------
  *I_B3_INT_CONTROL              ** IPG Controllo interno abilitato

***************************************
NoLSR_IPG_YLR:

LD   %config_machine28
EQ   2
JMPCN LSR_RAYCUS
      LD   I_LSR_READY
      ST   I_B1_LASER_READY              ** IPG Laser internal main power supply ON (Aux Power ON)

      LD   %PLCFLAGS.1
      ST   I_B7_LASER_ASSIGNED           ** IPG Laser ASSIGNED

	  LD   I_LSR_EMISSION_ON
      ST   I_B2_EMISSION_ON              ** IPG Emission ON

      LD   I_LSR_ASSIGNED
      ST   I_B8_POWER_SUPPLY             ** IPG power supply status

      LD   I_LSR_ERROR
      ST   I_B4_LASER_ERROR           ** IPG YLS YLR Laser in Alarm status
LSR_RAYCUS:

**************************************************
* nLight Resonator Management

PATH %Resonator[1]
PATH %LsrGest[0]

LD   %config_machine28
EQ   5
JMPCN no_nlight_resonator

LD   I_FW_READY_nLight
ST   I_I_FW_READY_nLight                     * NLIGHT: nLight ready to recieve input

LD   I_EMISS_nLight
ST   I_I_EMISS_nLight                        * NLIGHT: emiss nlight enable

LD   I_ERR_nLight
ST   I_I_ERR_nLight                          * NLIGHT: nlight error

LD   I_RDY_nLight
ST   I_I_RDY_nLight                          * NLIGHT: laser nlight ready

LD   I_ExtCtr_Ready_nLight
ST   I_I_ExtCtr_Ready_nLight                 * NLIGHT: nLight external control ready

no_nlight_resonator:

*************************************************
*   CAPACITIVE
*************************************************
PATH %Capacitive[0]

* Ingressi analogica
*----------------------------
* mainfast.plc
* LD   I_PREC_CAPACITIVO
* ST   IA_A18_19_DIST_LINEAR      * Capacitive sensor

* Ingressi digitali
*----------------------------

LD   %config_machine26
EQ   4
JMPC PREC_IO_TYPE

     LD   I_PREC_FAR
     ST   I_FAR_A10                  ** Far away

     LD   I_PREC_COLLISION
     ST   I_TIP_BODY_TOUCH_A11       ** Tip\Body Touch or Nozzle_Lost (TIP TOUCH:A11=1,A14=0,A15=0)

     LD   I_PREC_BROKEN
     ST   I_CABLE_CUT_A12            ** Cable cut

     LD   I_PREC_READY
     ST   I_READY_A13                ** Ready

     LD   I_PREC_BODY_TOUCH
     ST   I_BODY_TOUCH_A14           ** Body touch (A11=1,A14=1,A15=0)

     LD   I_PREC_REACH
     ST   I_NOZZLE_LOST_A15          ** Nozzle Lost/Pos reached (NOZZLE LOST:A11=1,A14=0,A15=1)

PREC_IO_TYPE:

LD   %config_machine26
EQ   4
JMPCN PREC_LIKE_ECAT

     LD   I_ECAT_FAR
     ST   I_FAR_A10                  ** Far away

     LD   I_ECAT_COLLISION
     ST   I_TIP_BODY_TOUCH_A11       ** Tip\Body Touch or Nozzle_Lost (TIP TOUCH:A11=1,A14=0,A15=0)

     LD   I_ECAT_BROKEN
     ST   I_CABLE_CUT_A12            ** Cable cut

     LD   I_ECAT_READY
     ST   I_READY_A13                ** Ready

     LD   I_ECAT_BODY_TOUCH
     ST   I_BODY_TOUCH_A14           ** Body touch (A11=1,A14=1,A15=0)

     LD   I_ECAT_REACH
     ST   I_NOZZLE_LOST_A15          ** Nozzle Lost/Pos reached (NOZZLE LOST:A11=1,A14=0,A15=1)

PREC_LIKE_ECAT:

*************************************************
*   LENS
*************************************************
PATH %Head_Laser[0]

*Gestione focale PRECITEC
***************************************
LD   %config_machine25
EQ   0
JMPCN NoLENS_PREC

  LDN  I_PREC_ERROR
  ST   I_I_PREC_ERROR                ** precitec in error

  LD   I_PREC_INPOS
  ST   I_I_PREC_POSITION_REACHED     ** Position Reached
***************************************
NoLENS_PREC:

END_FUNCTION

*******************************************************************************
*   I/O CONFIGURATION (OUTPUT)
*******************************************************************************
FUNCTION OUT_CONFIG

*************************************************
*   GENERIC
*************************************************
 *Uscite digitali
 *----------------------------
  LD  O_O_CNC_OK                  * CNC OK
  ST  O_CN_READY

 * LD  ALARM_ACT		         ** M100.3  Allarme attivo
 * ST  AlarmExt                    * Allarmi Esterno

* Hoerbiger Valve

*LD   O_O_ENAB_VALVE_HOERB
*ST   O_ENAB_VALVE_HOERB

LD   O_O_PILOT_HOERB
ST   O_PILOT_HOERB

LD   O_O_CALIB_REQ_HOERB
ST   O_CALIB_REQ_HOERB

LD   O_O_EV_OPEN_N2_HOERB
ST   O_EV_OPEN_N2_HOERB

LD   O_O_EV_OPEN_O2_HOERB
ST   O_EV_OPEN_O2_HOERB

LD   O_O_EV_OPEN_ARIA_HOERB
ST   O_EV_OPEN_ARIA_HOERB

*LD   O_O_GAS_ECAT_TYPE0_ENAB
*ST   O_GAS_ECAT_TYPE0_ENAB

LD   O_OA_GAS_HOERB
ST   OA_GAS_HOERB

*************************************************
*   GAS
*************************************************
 *Uscite analogica
 *----------------------------
 * LD  OA_GAS_ECAT_TYPE0           * Uscita Valvola Proporzionale Gas di taglio
 * ST  %ecat_ring0.EcatNode16.EcMDPOut1

 * LD  O_O_GAS_ECAT_TYPE0_ENAB     * Abilita Valvola Proporzionale
 * ST  %ecat_ring0.EcatNode16.EcMDPOut0.0

 *Uscite digitali
 *----------------------------
  LD  O_O_EV_ARIA_UGELLO         * Elettrovalvola aria ugello
  ST  O_EV_ARIA_UGELLO

  LD  O_O_EV_OPEN_ARIA           * Elettrovalvola apertura Aria taglio
  ST  O_EVGAS_ARIA

  LD  O_O_EV_OPEN_N2             * Elettrovalvola apertura Azoto
  ST  O_EVGAS_OAZOTO

  LD  O_O_EV_OPEN_O2             * Elettrovalvola apertura Ossigeno
  ST  O_EVGAS_OSSIGENO

  LD  O_O_EV_AUX_GAS             * Elettrovalvola ausiliaria (a valle della proporzionale)
  ST  O_EV_AUX_GAS

  LD  O_EVGAS_ARIA
  OR  O_EVGAS_OAZOTO
  OR  O_EVGAS_OSSIGENO
  ST  O_EVGAS_PRES                * Output pressurizzazione gas

 *SEGNALI NON GESTITI
 *----------------------------
  *O_O_EV_ASSISTENZA_TAGLIO      * Elettrovalvola assistenza taglio

*************************************************
*   RESONATOR
*************************************************
PATH %Resonator[0]
PATH %LsrGest[0]

*Gestione laser IPG YSL
***************************************
LD   %config_machine28
EQ   0
JMPCN NoLSR_IPG_YLS

 *Gestione yEmission direttamente su scheda PWM
 *----------------------------
 LD  OUT_isFlyCutModeON            * IN "FLYCUT" or M851 cannot write on this register
 JMPC YLS_FlyCut
  LD   O_A1_LASER_REQ             ** IPG Richiesta Laser
  ST   %QW911.8

  CAL  RTRIG_A1_LASER_REQ(CLK:=O_A1_LASER_REQ)
  CAL  TOF_A1_LASER_REQ(IN=RTRIG_A1_LASER_REQ.Q,PT=1000)

  LD   TOF_A1_LASER_REQ.Q
  ST   O_LSR_REQUEST
 YLS_FlyCut:

 *Uscite digitali
 *----------------------------
  LD   O_C1_LASER_SWITCH          ** IPG Laser Switch ON
  ST   O_LSR_LASER_ON

  LD   O_A4_LASER_RESET           ** IPG Resetta errori
  ST   O_LSR_RESET

  LD   O_A5_GUIDE_LASER           ** IPG Laser spot guide ON
  ST   O_LSR_GUIDE_ON

  LD   O_A6_ANALOG_CONTROL        ** IPG Controllo analogico ON
  ST   O_LSR_ANALOG_CONTROL

***************************************
NoLSR_IPG_YLS:

*Gestione laser IPG YSR - RACK
***************************************
LD   %config_machine28
EQ   1
JMPCN NoLSR_IPG_YLR

 *Gestione Remote start (solo IPG Rack)
 *----------------------------
  *Gestione fronte di salita
  *I_LSR_WORNING è collegato Laser PS Active Pin 5-7 conn.EMG)
*  CAL TM_OnLSR(IN=AuxOn,PT=500)
*  LD   TM_OnLSR.Q
*  AND  O_A1_LASER_REQ                ** IPG Richiesta Laser
*  ST   AppStartLSR
*  CAL  TM_StartButton(IN=AppStartLSR,PT=1500)

*  LD   TM_StartButton.Q
*  ST   O_LSR_REMOTE_START

 *Uscite digitali
 *----------------------------
  LD   O_A4_LASER_RESET           * IPG Resetta errori
  ST   O_LSR_RESET

  LD   O_A5_GUIDE_LASER           * IPG Laser spot guide ON
  ST   O_LSR_GUIDE_ON

***************************************
NoLSR_IPG_YLR:

LD   %config_machine28
EQ   2
JMPCN LSR_RAYCUS_OUT
      LD   O_A5_GUIDE_LASER           * IPG Laser spot guide ON
      ST   O_LSR_GUIDE_ON

      LD   O_A1_LASER_REQ
      ST   O_LSR_LASER_ON

	  LD   O_C1_LASER_SWITCH
	  ST   O_LSR_REMOTE_START

	  LD   O_A4_LASER_RESET           ** IPG Resetta errori
      ST   O_LSR_RESET

	  * Some models of Raycus needs to add delay with fc-out (Laser Enable)
	  * In such a case, it requires to use pure PWM control and FcOut always 1
	  LD   PAR_combinedMode
	  JMPCN RAY_PUREPWM
	       LD   O_A1_LASER_REQ             ** IPG Richiesta Laser
           ST   %QW911.8
	  RAY_PUREPWM:
LSR_RAYCUS_OUT:

**************************************************
* nLight Resonator Management

PATH %Resonator[1]
PATH %LsrGest[0]

LD   %config_machine28
EQ   5
JMPCN no_nlight_resonator1

LD   O_O_EXTEN_IN_nLight                   * NLIGHT: nlight exten in
ST   %M5.0

LD   O_O_GUIDE_nLight                      * NLIGHT: Guide laser nlight
ST   O_LSR_GUIDE_ON

*LD   O_O_SYSTEM_ON_nLight                  * NLIGHT: nlight system on
*ST   %QW3.3

LD   O_O_RESET_nLight                      * NLIGHT: reset error nlight
ST   O_LSR_RESET

LD   O_O_ExtCtr_ENABLE_nLight              * NLIGHT: Enable external control of nlight
ST   %M5.0

no_nlight_resonator1:

*************************************************
*   CAPACITIVE
*************************************************
PATH %Capacitive[0]
 *Uscite digitali
 *----------------------------

LD   %config_machine26
EQ   4
JMPC PREC_IO_TYPE_OUT

     LD  O_CALIBRA_REQ_A3            * Calibration request
     ST  O_PREC_CALIBRAZIONE

     LD  O_STROBE_A7                 * Strobe
     ST  O_PREC_STROBE

     LD  O_SELCHAR_BIT0_A4           * Selecting the calibrated characteristic curve (1-8)
     ST  O_PREC_SELCHAR_0

     LD  O_SELCHAR_BIT1_A5           * Selecting the calibrated characteristic curve (1-8)
     ST  O_PREC_SELCHAR_1

     LD  O_SELCHAR_BIT2_A6           * Selecting the calibrated characteristic curve (1-8)
     ST  O_PREC_SELCHAR_2

PREC_IO_TYPE_OUT:

LD   %config_machine26
EQ   4
JMPCN PREC_LIKE_ECAT_OUT

     LD  O_CALIBRA_REQ_A3            * Calibration request
     ST  O_ECAT_CALIBRAZIONE

     LD  O_STROBE_A7                 * Strobe
     ST  O_ECAT_STROBE

     LD  O_SELCHAR_BIT0_A4           * Selecting the calibrated characteristic curve (1-8)
     ST  O_ECAT_SELCHAR_0

     LD  O_SELCHAR_BIT1_A5           * Selecting the calibrated characteristic curve (1-8)
     ST  O_ECAT_SELCHAR_1

     LD  O_SELCHAR_BIT2_A6           * Selecting the calibrated characteristic curve (1-8)
     ST  O_ECAT_SELCHAR_2

PREC_LIKE_ECAT_OUT:

*************************************************
*   LENS
*************************************************
PATH %Head_Laser[0]

*Gestione focale PRECITEC
***************************************
LD   %config_machine25
EQ   0
JMPCN NoLENS_PREC

  LD   O_O_PREC_AUTOMATIC         * Automatic request fo precitec head
  ST   O_PREC_POSITION

  LD   O_O_PREC_REFERENCE         * Reference signal for precitec head
  ST   O_PREC_REF

  LD   OA_FOCALE                  * Focal analog out
  ST   O_PREC_FOCALE

***************************************
NoLENS_PREC:

*************************************************
*   Clamp
*************************************************

LD   O_O_CLAMP_C_CLOSE           *AT %M62.9;
ST   O_CLAMP_C_CLOSE

LD   O_O_CLAMP_C_OPEN           *AT %M62.10;
ST   O_CLAMP_C_OPEN

LD   O_O_CLAMP_C1_CLOSE           *AT %M62.11;
ST   O_CLAMP_C1_CLOSE

LD   O_O_CLAMP_C1_OPEN           *AT %M62.12;
ST   O_CLAMP_C1_OPEN

*************************************************
*   MACHINE LIGHT
*************************************************
LD   O_O_LUCE_CABINA          * AT %M60.0;
ST   O_LUCE_CABINA

LD   O_O_LAMPADA_ROSSA
ST   O_LAMPADA_ROSSA

LD   O_O_LAMPADA_ROSSA
AND  %PLCFLAGS.10
ANDN %LSRPlcOp1.27
ST   O_BUZZER_ALARM

LD   O_O_LAMPADA_ARANCIONE
ST   O_LAMPADA_ARANCIONE

LD   O_O_LAMPADA_VERDE
ST   O_LAMPADA_VERDE

LD   O_O_BUZZER_START_CIC
ST   O_BUZZER_START_CIC

*************************************************
*   Lubrication
*************************************************
LD   I_LUB_LOW_LEVEL
ST   I_I_LUB_LOW_LEVEL        *AT %M55.5;

LD   I_LUB_LOW_PRESSURE
ST   I_I_LUB_LOW_PRESSURE     *AT %M55.9;

LD   I_OVER_PRES_LUB
ST   I_I_OVER_PRES_LUB        *AT %M55.10

LD   O_O_LUB                  *AT %M60.7;
ST   O_LUB

*************************************************
*   ASPIRATORE
*************************************************

LD   O_START_ASPIRATORE        *AT %DigOutAspirator1.0  Command START for Aspiration system
ST   START_ASPIRATORE
ST   START_ASPIRATORE_FUMI

*************************************************
*   Limit Switch
*************************************************

LD   I_FC_Y1_POS
ST   I_I_FC_Y1_POS        *AT %M53.2;

LD   I_FC_Y1_NEG
ST   I_I_FC_Y1_NEG        *AT %M53.3;

LD   I_FC_X1_POS
ST   I_I_FC_X1_POS        *AT %M53.0;

LD   I_FC_X1_NEG
ST   I_I_FC_X1_NEG        *AT %M53.1;

LD   I_FC_Z1_POS
ST   I_I_FC_Z1_POS        *AT %M53.4;

LD   I_FC_Z1_NEG
ST   I_I_FC_Z1_NEG        *AT %M53.5;

LD   I_FC_UV_POS
ST   I_I_FC_UV_POS        *AT %M53.6;

LD   I_FC_UV_NEG
ST   I_I_FC_UV_NEG        *AT %M53.7;

LD   I_FC_W1_POS
ST   I_I_FC_W1_POS        *AT %M53.8;

LD   I_FC_W1_NEG
ST   I_I_FC_W1_NEG        *AT %M53.9;

LD   I_FC_V_POS
ST   I_I_FC_V_POS         *AT %M53.18;

LD   I_FC_V_NEG
ST   I_I_FC_V_NEG         *AT %M53.19;

LD   I_FC_Z1_SUP_NEG
ST   I_I_FC_Z1_SUP_NEG

LD   I_FC_Z2_SUP_NEG
ST   I_I_FC_Z2_SUP_NEG

LD   I_FC_Z3_SUP_NEG
ST   I_I_FC_Z3_SUP_NEG

LD   I_FC_Z4_SUP_NEG
ST   I_I_FC_Z4_SUP_NEG

LD   I_FC_Z1_SUP_POS
ST   I_I_FC_Z1_SUP_POS

LD   I_FC_Z2_SUP_POS
ST   I_I_FC_Z2_SUP_POS

LD   I_FC_Z3_SUP_POS
ST   I_I_FC_Z3_SUP_POS

LD   I_FC_Z4_SUP_POS
ST   I_I_FC_Z4_SUP_POS

LD   I_FC_L1_NEG
ST   I_I_FC_L1_NEG

LD   I_FC_L2_NEG
ST   I_I_FC_L2_NEG

LD   I_FC_L3_NEG
ST   I_I_FC_L3_NEG

LD   I_FC_L4_NEG
ST   I_I_FC_L4_NEG

LD   I_FC_L5_NEG
ST   I_I_FC_L5_NEG

LD   I_FC_L1_POS
ST   I_I_FC_L1_POS

LD   I_FC_L2_POS
ST   I_I_FC_L2_POS

LD   I_FC_L3_POS
ST   I_I_FC_L3_POS

LD   I_FC_L4_POS
ST   I_I_FC_L4_POS

LD   I_FC_L5_POS
ST   I_I_FC_L5_POS

LD   I_FC_O4_POS
ST   I_I_FC_O4_POS
LD   I_FC_O3_POS
ST   I_I_FC_O3_POS
LD   I_FC_O2_POS
ST   I_I_FC_O2_POS
LD   I_FC_O1_POS
ST   I_I_FC_O1_POS

LD   I_FC_O4_NEG
ST   I_I_FC_O4_NEG
LD   I_FC_O3_NEG
ST   I_I_FC_O3_NEG
LD   I_FC_O2_NEG
ST   I_I_FC_O2_NEG
LD   I_FC_O1_NEG
ST   I_I_FC_O1_NEG

LD   I_FC_W_NEG
ST   I_I_FC_W_NEG
LD   I_FC_W_POS
ST   I_I_FC_W_POS

LD   I_FC_B1_POS
ST   I_I_FC_B1_POS
LD   I_FC_B1_NEG
ST   I_I_FC_B1_NEG

LDN  I_AntiColide_1
ORN  I_AntiColide_2
ST   I_I_AntiColide
S    %PLCerr21.24

*****************************************************
*   Proportional valves type 2
*   ---> N2, AIR share the same valve (0-10v,1-5v)
*   ---> O2 (0-10v,1-5v)
*   ---> Feedback to use always inputs on CNC (4095)
*****************************************************
LD   %config_machine29             ** Proportional valve manage only with OXYGEN
EQ   2
JMPCN AIRO2_O2_SMCS

LD   0
ST   O_OA_GAS_2
ST   O_OA_GAS

LD   819
ST   IA_Feedback_GAS_OUT

LD   O_O_EV_OPEN_ARIA
OR   O_O_EV_OPEN_N2
JMPCN NO_HP_VALVE

LD   OA_GAS
ST   O_OA_GAS
LD   0
ST   O_OA_GAS_2

LD   I_IA_Feedback_GAS_OUT
ST   IA_Feedback_GAS_OUT

NO_HP_VALVE:

LD   O_O_EV_OPEN_O2
JMPCN NO_LP_VALVE

LD   0
ST   O_OA_GAS
LD   OA_GAS
ST   O_OA_GAS_2

LD   I_IA_Feedback_GAS_OUT_O2
ST   IA_Feedback_GAS_OUT

NO_LP_VALVE:

AIRO2_O2_SMCS:

*************************************************
* SAFETY DEVICE
*************************************************
LD   DoorSafety
EQ   0
JMPCN NOSFTDOOR
LD   0
ST   O_Unlock_Fence
ST   O_O_Guard_Door_1
ST   O_O_Guard_Door_2
NOSFTDOOR:

LD   DoorSafety
EQ   1
JMPCN SAFETYDOOR_1
     LD   PRGRUN_CN0
     ANDN PRGSTOP_CN0
     STN   O_Lock_Safety_Door
     ST  O_Safety_Bypass

     LDN  I_SAFETY_DOOR
     AND  PRGRUN_CN0
     S    %PLCerr21.15            ** Machine Door Open

    * LDN  I_Grating_Alm
    * AND  PRGRUN_CN0
    * ANDN I_SafetyDevice_Bypass
    * S    %PLCerr21.16            ** Laser Safe Activated
    *
    * CAL  TP_Fence(IN=I_UnlckFence_Btn,PT=3000)
    * LD   TP_Fence.Q
    * AND  %PLCFLAGS.10
    * OR   O_Unlock_Fence
    * ST   O_Unlock_Fence_LED
    *
    * CAL  FTRIG_Fence(CLK=TP_Fence.Q)
    * LD   FTRIG_Fence.Q
    * S    O_Unlock_Fence
    *
    * LD   O_Unlock_Fence
    * OR   TP_Fence.Q
    * AND   PRGRUN_CN0
    * S    %PLCerr21.17
SAFETYDOOR_1:

LD   DoorSafety
EQ   2
JMPCN SAFETYDOOR_2
     LD   EnAutoDoor
     AND  %cn0.rc8.0
	 ST   GuardDoorAutoUp

	 LD   iso_G580_Running
	 AND  %cn0.rc8.0
	 ST   GuardDoorAutoDwn

     CAL  R_TRIG_Door_Up_Gui_1(CLK=Door1_Up_Gui)
	 LD   R_TRIG_Door_Up_Gui_1.Q          ** (LsGui0.17)
	 OR   GuardDoorAutoUp
     S 	  O_O_Guard_Door_1

     CAL  R_TRIG_Door_Down_Gui_1(CLK=Door1_Down_Gui)
     LD   R_TRIG_Door_Down_Gui_1.Q
	 OR   GuardDoorAutoDwn
     R    O_O_Guard_Door_1

     CAL  R_TRIG_Door_Up_Gui_2(CLK=Door2_Up_Gui)
	 LD   R_TRIG_Door_Up_Gui_2.Q          ** (LsGui0.19)
	 OR   GuardDoorAutoUp
     S 	  O_O_Guard_Door_2

  	 CAL  R_TRIG_Door_Down_Gui_2(CLK=Door2_Down_Gui)
     LD   R_TRIG_Door_Down_Gui_2.Q
	 OR   GuardDoorAutoDwn
     R    O_O_Guard_Door_2
SAFETYDOOR_2:

LD   Pul_Reset              ** (gPlc0.3)Reset pushbutton
ST   O_RESET_SAFETY_DEVICE
R    %PLCerr21.15           ** Machine Door Open
R    %PLCerr21.16            ** Laser Safe Activated
R    %PLCerr21.17
R    %PLCerr21.24
R    O_Unlock_Fence

LD   O_O_Guard_Door_1
ST   O_Guard_Door_1
STN  O_Guard_Door_1_Dwn

LD   O_O_Guard_Door_2
ST   O_Guard_Door_2
STN  O_Guard_Door_2_Dwn

END_FUNCTION
